TEXTLIST TextList_CryoPump
  54 = 'Trame Manuelle' | FR: 'Trame Manuelle' | EN: 'Manual Frame'
  55 = 'paramètres de régénération' | FR: 'Paramètres de régénération' | EN: 'Regeneration settings'
  56 = '' | FR: 'Pompe Cryo' | EN: 'Cryo pump'
  3 = '' | FR: 'Forçage' | EN: 'Forcing'
  4 = '' | FR: 'Etat de la pompe' | EN: 'Pump Status'
  5 = '' | FR: 'Température du 1er étage (°K)' | EN: '1st stage temperature (°K)'
  6 = '' | FR: 'Température du 2ème étage (°K)' | EN: '2nd stage temperature (°K)'
  8 = 'Activé' | FR: 'Pompe activée' | EN: 'Pump activated'
  7 = 'Désactivé' | FR: 'Pompe désactivée' | EN: 'Pump disabled'
  9 = '' | FR: 'Retour' | EN: 'Back'
  10 = '' | FR: 'Temps de balayage long (min)' | EN: 'Extended purge time (min)'
  11 = '' | FR: 'Délai de redémarrage (h)' | EN: 'Delay restart (h)'
  12 = '' | FR: 'Nombre de cycles de balayage' | EN: 'Repurge cycles'
  13 = '' | FR: 'Temps de cycle du balayage (min)' | EN: 'Repurge time (min)'
  14 = '' | FR: 'Nombre de cycles de remontée en pression' | EN: 'Rate of rise cycles'
  15 = '' | FR: 'Sous pression' | EN: 'Rough to pressure'
  16 = '' | FR: "Verrouillage de la vanne d'arrêt" | EN: 'Rough Valve Interlock'
  17 = '' | FR: 'Température de démarrage (°K)' | EN: 'Start Up Temperature (°K)'
  18 = '' | FR: 'Lecture des paramètres enregistrés dans la pompe' | EN: 'Reading parameters stored in the pump'
  19 = '' | FR: 'Ecriture des paramètres dans la pompe' | EN: 'Writing parameters to the pump'
  20 = '' | FR: 'Lancer la régénération ' | EN: 'Launch regeneration '
  21 = '' | FR: 'Stopper la régénération ' | EN: 'Stop regeneration '
  22 = '' | FR: 'Commande :' | EN: 'Command :'
  23 = '' | FR: 'Réponse :' | EN: 'Response :'
  24 = '' | FR: 'Envoie Trame ' | EN: 'Send Frame'
  25 = '' | FR: 'Pompe Cryo On-Board' | EN: 'CryoPump On-Board'
  26 = '' | FR: 'ÉCHAUFFEMENT' | EN: 'WARM-UP'
  27 = '' | FR: 'DÉFAILLANCE DU GAZ DE PURGE' | EN: 'PURGE GAS FAILURE'
  28 = '' | FR: 'Balayage long' | EN: 'Extended purge'
  29 = '' | FR: 'Pression de pompage primaire (μ)' | EN: 'Rough to base pressure (μ)'
  30 = '' | FR: 'Remontée en pression ROR (μ/min)' | EN: 'Rate of rise ROR (μ/min)'
  31 = '' | FR: 'REFROIDISSEMENT' | EN: 'COOLDOWN'
  32 = '' | FR: 'DÉLAI DE REDÉMARRAGE' | EN: 'DELAY RESTART'
  33 = '' | FR: 'DÉLAI DE DÉMARRAGE' | EN: 'DELAY START'
  34 = '' | FR: 'RÉGÉNÉRATION TERMINÉE' | EN: 'REGEN COMPLETED'
  35 = '' | FR: 'RÉGÉNÉRATION ARRÊTÉE' | EN: 'REGEN ABORTED'
  36 = '' | FR: "Retour aux paramètres d'usine" | EN: 'Return to factory settings'
  38 = '' | FR: 'Ouverte' | EN: 'Open'
  37 = '' | FR: 'Fermé' | EN: 'Close'
  39 = '' | FR: 'Etat de la vanne primaire' | EN: 'Rough Valve Status'
  40 = '' | FR: 'Etat de la vanne de balayage' | EN: 'Purge Valve Status'
  41 = '' | FR: 'Vanne primaire' | EN: 'Rough Valve'
  42 = '' | FR: 'Vanne de balayage' | EN: 'Purge Valve'
  43 = '' | FR: 'Etapes de la régénération en cours :' | EN: 'Stages of regeneration in progress :'
  44 = '' | FR: 'Cryo éteinte' | EN: 'Cryo Off'
  45 = '' | FR: 'Rétablissement après coupure' | EN: 'Power Fail Recovery'
  46 = '' | FR: 'Informations de la pompe' | EN: 'Pump Infos'
  47 = '' | FR: 'Numéro de série de la pompe' | EN: 'Pump Serial Number'
  48 = '' | FR: 'Nombre de cycles de régénération completés' | EN: 'Number of complete regeneration'
  49 = '' | FR: 'Temps depuis la dernière régénération (h)' | EN: 'Time since last regeneration (h)'
  50 = '' | FR: 'Niveau de révision du logiciel' | EN: 'Software revision level'
  51 = '' | FR: 'Temps de fonctionnement de la pompe (h)' | EN: 'Pump operating time (h)'
  52 = '' | FR: 'Réinitialiser ' | EN: 'RESET'
  53 = '' | FR: 'Pression (μ)' | EN: 'Pressure (μ)'
  0 = '' | FR: 'OFF' | EN: 'OFF'
  1 = '' | FR: 'ON' | EN: 'ON'
  2 = '' | FR: 'COOL' | EN: 'COOL'
  57 = '' | FR: 'Délai de démarrage (h)' | EN: 'Delay start (h)'
  58 = '' | FR: "TEMPS D'ÉCHAUFFEMENT" | EN: 'WARMUP TIMEOUT'
  59 = '' | FR: 'AUCUNE ERREUR' | EN: 'NO ERROR'
  60 = '' | FR: 'DÉLAI DE REFROIDISSEMENT' | EN: 'COOLDOWN TIMEOUT'
  61 = '' | FR: 'ERREUR DANS LE ROR' | EN: 'ERROR IN ROR'
  62 = '' | FR: 'LA LIMITE DE CYCLES ROR A ÉTÉ ATTEINTE' | EN: 'ROR CYCLE LIMIT WAS REACHED'
  63 = '' | FR: 'ARRÊT MANUEL' | EN: 'MANUAL ABORT'
  64 = '' | FR: "DÉLAI D'ATTENTE DE LA VANNE PRIMAIRE" | EN: 'ROUGH VALVE TIMEOUT'
  65 = '' | FR: 'BOGUE DU SYSTÈME' | EN: 'SYSTEM BUG'
  66 = '' | FR: 'Numero du relais :' | EN: 'Relay number :'
  67 = '' | FR: 'Commande du paramètre :' | EN: 'Settings command :'
  68 = '' | FR: 'Valeur :' | EN: 'Value :'
  69 = '' | FR: 'Appliquer ces paramètres' | EN: 'Apply this settings'
  70 = '' | FR: 'Température du 1er étage' | EN: '1st stage temperature'
  71 = '' | FR: 'Température de 2ème étage' | EN: '2nd stage temperature'
  72 = '' | FR: 'Pression Cryo TC' | EN: 'Cryo TC pressure'
  73 = '' | FR: 'Pression TC auxiliaire' | EN: 'Aux TC pressure'
  74 = '' | FR: "Délai d'attente (passage ON/OFF)" | EN: 'Time delay (switch ON/OFF)'
  75 = '' | FR: 'Fonction manuelle = ON' | EN: 'Manual Function = ON'
  76 = '' | FR: 'Fonction manuelle = OFF' | EN: 'Manual Function = OFF'
  77 = '' | FR: "Suivi de l'état de régénération" | EN: 'Regen track'
  78 = '' | FR: "Suivi de l'état de vanne primaire" | EN: 'Rough valve track'
  79 = '' | FR: "Suivi de l'état de la pompe cryo" | EN: 'Cryopump track'
  80 = '' | FR: 'Paramétrages des relais' | EN: 'Relay settings'
  81 = '' | FR: 'Mode manuel' | EN: 'Manual mode'
  82 = '' | FR: 'Mode automatique' | EN: 'Automatic mode'
  84 = '' | FR: 'Relais actif (ON)' | EN: 'Enable relay (ON)'
  83 = '' | FR: 'Relais inactif (OFF)' | EN: 'Disable relay (OFF)'
  85 = '' | FR: 'Restaure les paramètres automatiques' | EN: 'Restores automatic settings'
  86 = '' | FR: 'Cycle de rebalayage' | EN: 'Repurge cycle'
  1000 = '' | FR: 'Pas de données' | EN: 'No data'
  87 = '' | FR: 'Informations supplémentaires' | EN: 'Further information'
  88 = '' | FR: 'Lecture ' | EN: 'Read'
  89 = '' | FR: 'Attention !' | EN: 'Warning !'
  90 = '' | FR: 'Cette action peut altérer le bon fonctionnement de la machine. Voulez-vous continuer ?' | EN: "This action may affect the machine's operation. Do you want to continue?"
  91 = '' | FR: "Êtes-vous sûr de retourner aux paramètres d'usine ?" | EN: 'Are you sure you want to return to factory settings ?'
  92 = '' | FR: 'Confirmer' | EN: 'Confirm'
  93 = '' | FR: 'Annuler' | EN: 'Cancel'
  94 = '' | FR: 'Etats' | EN: 'States'
  95 = '' | FR: 'Fermé' | EN: 'Closed'
  96 = '' | FR: 'Régulation de la température du 1er étage' | EN: '1st floor temperature control'
  97 = '' | FR: 'maintenance alliance concept' | EN: 'alliance concept maintenance'
  98 = '' | FR: 'Configuration de la pompe cryo' | EN: 'Cryo pump settings'
   = ''
END_TEXTLIST

(* stored: Version 1.1.0.1, ProductVersion 3.1.4026.18
   TextList TextList_CryoPump: Id {224b41d9-2649-4cbc-982e-7290163048b1} *)
